% RSLogix 500 project P3.RSS, saved by version 12.00.00.00 %
PROJECT "UNTITLED"    % processor: type code 162 %

PROGRAM FILES
  LAD 2   6 rungs

DATA FILES
  S2 STATUS  83 elements
  B3 BINARY  1 elements
  T4 TIMER  1 elements
  C5 COUNTER  1 elements
  R6 CONTROL  1 elements
  N7 INTEGER  5 elements
  F8 FLOAT  1 elements
  ST9 STR  12 elements

LADDER 2
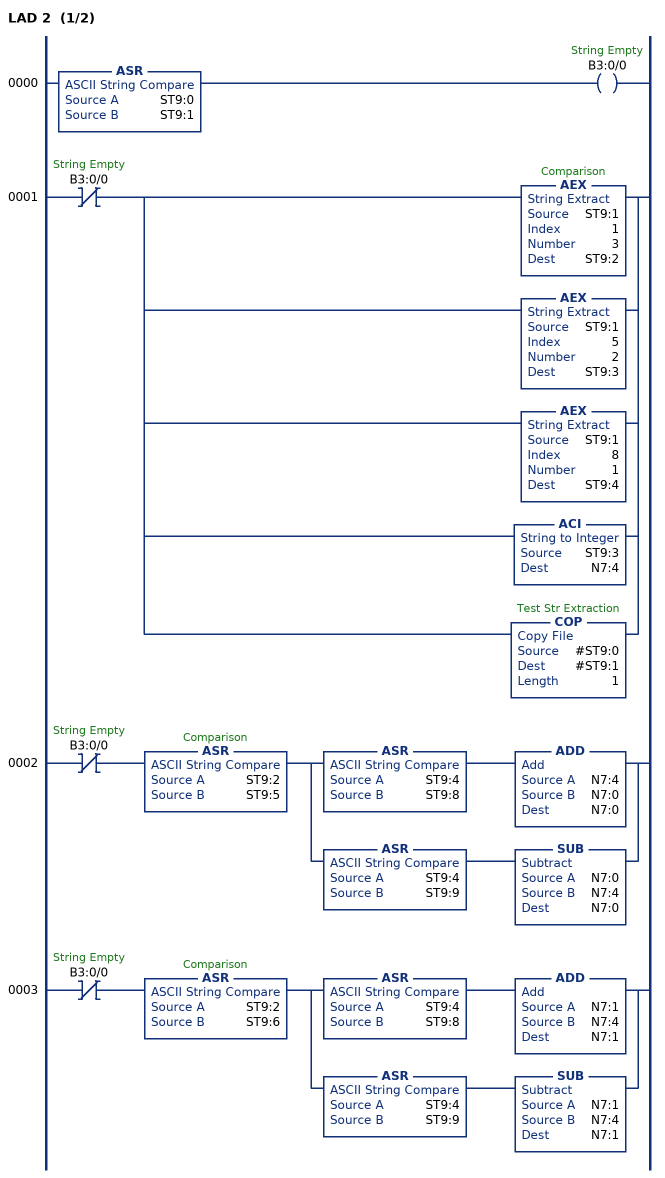
% Rung: 0 %
SOR ASR ST9:0 ST9:1 OTE B3:0/0 EOR
%   ST9:1  "Test Str Extraction" %
%   B3:0/0  "String Empty" %
% Rung: 1 %
SOR XIO B3:0/0 BST AEX ST9:1 1 3 ST9:2 NXB AEX ST9:1 5 2 ST9:3 NXB AEX ST9:1 8 1 ST9:4 NXB ACI ST9:3 N7:4 NXB COP #ST9:0 #ST9:1 1 BND EOR
%   B3:0/0  "String Empty" %
%   ST9:1  "Test Str Extraction" %
%   ST9:2  "Comparison" %
% Rung: 2 %
SOR XIO B3:0/0 ASR ST9:2 ST9:5 BST ASR ST9:4 ST9:8 ADD N7:4 N7:0 N7:0 NXB ASR ST9:4 ST9:9 SUB N7:0 N7:4 N7:0 BND EOR
%   B3:0/0  "String Empty" %
%   ST9:2  "Comparison" %
% Rung: 3 %
SOR XIO B3:0/0 ASR ST9:2 ST9:6 BST ASR ST9:4 ST9:8 ADD N7:1 N7:4 N7:1 NXB ASR ST9:4 ST9:9 SUB N7:1 N7:4 N7:1 BND EOR
%   B3:0/0  "String Empty" %
%   ST9:2  "Comparison" %

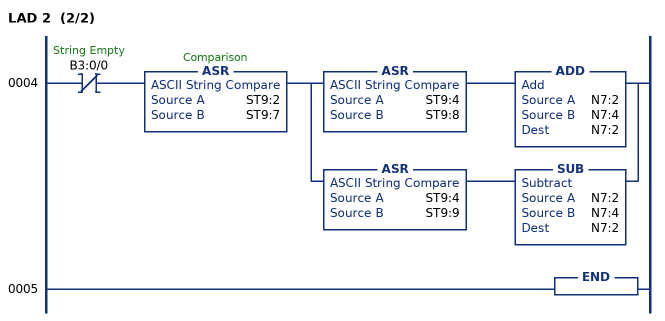
% Rung: 4 %
SOR XIO B3:0/0 ASR ST9:2 ST9:7 BST ASR ST9:4 ST9:8 ADD N7:2 N7:4 N7:2 NXB ASR ST9:4 ST9:9 SUB N7:2 N7:4 N7:2 BND EOR
%   B3:0/0  "String Empty" %
%   ST9:2  "Comparison" %
% Rung: 5 %
SOR END EOR

OTHER DOCUMENTED ADDRESSES
  B3:0/1  "ONS"
  B3:0/2  "ONS2"

DATA TABLE (non-zero values as saved)
DATA B3
% B3:0 % 0X0001
DATA N7
% N7:0 % 0 10 30 0 20
DATA ST9
% ST9:0 % "0"
% ST9:1 % "0"
% ST9:2 % "789"
% ST9:3 % "20"
% ST9:4 % "2"
% ST9:5 % "123"
% ST9:6 % "456"
% ST9:7 % "789"
% ST9:8 % "1"
% ST9:9 % "2"
